FUNCTION_BLOCK FB_Integrator
VAR_INPUT
	u_k		: REAL;
	T		: REAL;
END_VAR
VAR_OUTPUT
	y_k		: REAL;
END_VAR
VAR
	y_k_1	: REAL;
END_VAR

y_k := u_k * T + y_k_1;
y_k_1 := y_k;

END_FUNCTION_BLOCK

(* stored: Version 1.1.0.1, ProductVersion 3.1.4024.9
   POU FB_Integrator: Id {d2a5d47a-22c8-4def-a768-73763ee1c5c1}, SpecialFunc None *)
